Fanuc KAREL source: SET_PERCH.kl

PROGRAM T
%NOLOCKGROUP
VAR
 v0 : JOINTPOS
 v1 : ARRAY[6] OF REAL
 v2 : INTEGER
BEGIN
 SET_PERCH(v0, v1, v2)
END T
